Fanuc TP program (LS listing): BEND.LS

/PROG  BEND
/ATTR
OWNER		= MNEDITOR;
COMMENT		= "";
PROG_SIZE	= 376;
CREATE		= DATE 25-09-03  TIME 10:33:30;
MODIFIED	= DATE 26-01-14  TIME 20:07:16;
FILE_NAME	= PINCH;
VERSION		= 0;
LINE_COUNT	= 13;
MEMORY_SIZE	= 828;
PROTECT		= READ_WRITE;
STORAGE		= SHADOW;
TCD:  STACK_SIZE	= 0,
      TASK_PRIORITY	= 50,
      TIME_SLICE	= 0,
      BUSY_LAMP_OFF	= 0,
      ABORT_REQUEST	= 0,
      PAUSE_REQUEST	= 0;
DEFAULT_GROUP	= 1,*,*,*,*;
CONTROL_CODE	= 00000000 00000000;
LOCAL_REGISTERS	= 0,0,0;
/APPL

AUTO_SINGULARITY_HEADER;
  ENABLE_SINGULARITY_AVOIDANCE   : TRUE;

LINE_TRACK;
  LINE_TRACK_SCHEDULE_NUMBER      : 0;
  LINE_TRACK_BOUNDARY_NUMBER      : 0;
  CONTINUE_TRACK_AT_PROG_END      : TRUE;

/MN
   1:  IF (DI[25:RB_TANDEM]=OFF),JMP LBL[1] ;
   2:  WAIT (DO[22:Pinch_Latch])    ;
   3:  DO[27:RB_PEDALDN]=ON ;
   4:  DO[22:Pinch_Latch]=OFF ;
   5:  JMP LBL[2] ;
   6:   ;
   7:  LBL[1] ;
   8:   ;
   9:  UALM[5] ;
  10:   ;
  11:  PAUSE ;
  12:   ;
  13:  LBL[2] ;
/POS
/END
